(*********************************** G.D S.p.A. - Technical Department ***********************************
============= PROGRAM INFO ============
FOLDER:             TBD
MACHINES INVOLVED:  TBD 

============= DESCRIPTION =============

============= REVISIONS ===============
Date		Version	 	Author      	Description             
----------	-------		------------  	--------------------------------------------
2019/04/24 	0000.00	 	M.Grasso		Creation of the PRG

**********************************************************************************************************)
(*$R 
	process_ref:= prc; 
$*)
PROGRAM csp_main_safety_drives
VAR
	prc:					process;
	prc_path:				STRING;	
END_VAR

_read_var_input();

_objects_manager();

IF NOT objects_running()
THEN
	RETURN;	
END_IF

_read_process_image();

_mode_manager();

CASE process_get_mode(prc) OF
	MODE_ABSENT,
	MODE_INACTIVE:
		RETURN;
	MODE_TEST:
		;
END_CASE

_set_runtime_properties();

(********************************* BODY *********************************)

(************************************************************************)

_handle_messages();

_write_output();

ACTION _handle_messages:
;
END_ACTION

ACTION _handle_process_test:
;
END_ACTION

ACTION _mode_manager:
IF process_mode_req_is_pending(prc)
THEN
    process_apply_mode_req_first_step(prc);
    CASE process_get_mode(prc) OF
        MODE_TO_ABSENT:
			;
        MODE_TO_INACTIVE:
			;
        MODE_TO_TEST:
			;
        MODE_TO_OPERATIONAL:
			;
    END_CASE
    process_apply_mode_req_second_step(prc);
END_IF
END_ACTION

ACTION _objects_manager:
IF objects_initialization()
THEN
	sub_process_init(
		object_name					:= 'csp_main_safety_drives.prc', 
		process						:= csp_main_safety.prc, 
		CONVERSION_this				:= prc);
		
	prc_path 						:= process_get_path(prc);		
END_IF

IF objects_running()
THEN
	process_cycle(prc);
END_IF
END_ACTION

ACTION _read_process_image:
;
END_ACTION

ACTION _read_var_input:
;
END_ACTION

ACTION _set_runtime_properties:
;
END_ACTION

ACTION _write_output:
;
END_ACTION

END_PROGRAM

(* stored: Version 1.1.0.1, ProductVersion 3.1.4022.12
   POU csp_main_safety_drives: Id {32eb667d-678b-44a9-b776-f1b11cd3dfd7}, SpecialFunc None
   Action _handle_messages: Id {71b7fe4d-91b5-4d8c-8263-6d5386173ffb}
   Action _handle_process_test: Id {5bfb6953-1b49-4bc6-90b2-df8742528a3b}
   Action _mode_manager: Id {720cf2e6-339e-439f-a4f1-d18c9455eb13}
   Action _objects_manager: Id {f2f1d613-4fde-4ef7-92d5-03c8e4cc3662}
   Action _read_process_image: Id {93dd134b-0036-4f4e-a825-782e23102221}
   Action _read_var_input: Id {235fcacf-734e-4854-845f-63ff00d5412f}
   Action _set_runtime_properties: Id {7bf5bf0a-2168-4a3a-b869-8284d71e4a7d}
   Action _write_output: Id {eba58ed0-a546-4825-aa60-156f9fde5b73} *)
